// TIA Portal V20 export
FUNCTION "Mode_C3" : Void   // FC3, LAD
// stored: Access Published, IsIECCheckEnabled true, Namespace C3, SetENOAutomatically false
   VAR_INPUT
      on : Bool;
      off : Bool;
   END_VAR
   VAR_IN_OUT
      mode : Bool;
   END_VAR
BEGIN

REGION Network 1
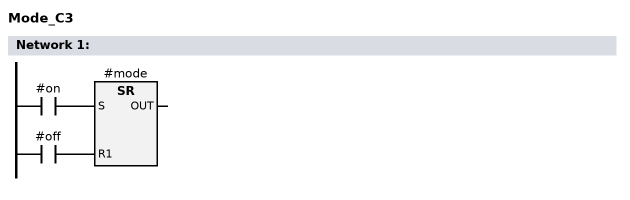
   RUNG wire#powerrail
      Contact( #on )
      S_SR(operand := #mode, r1 := wire#w1)
   END_RUNG
   RUNG wire#powerrail
      Contact( #off )
   END_RUNG wire#w1
   // the same network as SCL:
   IF #on THEN
       #mode := TRUE;   // SR flip-flop
   END_IF;
   IF #off THEN #mode := FALSE; END_IF;
END_REGION
END_FUNCTION
